PROGRAM ModeControl
VAR
	AutoModeButtonClick: BOOL;
	AutoMode: BOOL;
	ManualModeButtonClick: BOOL;
	ManualMode: BOOL;
END_VAR

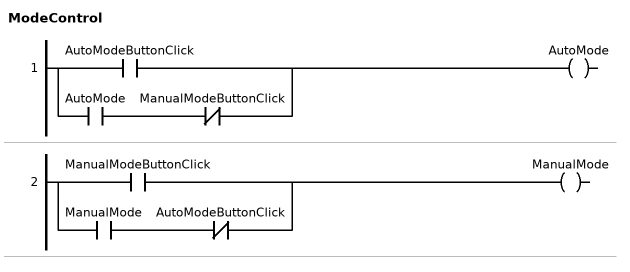
// NETWORK 1
AutoMode := AutoModeButtonClick OR AutoMode AND NOT ManualModeButtonClick;

// NETWORK 2
ManualMode := ManualModeButtonClick OR ManualMode AND NOT AutoModeButtonClick;

END_PROGRAM

(* stored: Version 1.1.0.1, ProductVersion 3.1.4024.12
   POU ModeControl: Id {e24a47d9-e45f-4121-9c79-84f0e558d7dd}, SpecialFunc None *)
